Staubli VAL3: stop.pgx

program stop()
begin
  popUpMsg("Press CS8 to get back to Main Menue")
  resetMotion()
end
